{attribute 'qualified_only'}
{attribute 'strict'}
{attribute 'to_string'}
TYPE ACTIVITY_STOPPING_STATE :
(
	WORK_IN_PROGRESS := 0,
	WORK_STOPPED,
	WORK_COMPLETED,
	WORK_HALTED
);
END_TYPE

(* stored: Version 1.1.0.1
   DUT ACTIVITY_STOPPING_STATE: Id {897ba669-f421-4703-a7fe-d511c03a2d21} *)
